Universal Robots PolyScope program: AG_touchoff_demo_tcp.urp

Program AG_touchoff_demo_tcp (installation=AutoGrind directory=/programs/AutoGrind createdIn=5.9.1.1031110 lastSavedIn=5.9.1.1031110 robotSerialNumber=20195501059)
Calibrated DH parameters: a=[0.000146, -0.418764, -0.053981, 0.000058, -0.000023, 0]; d=[0.162545, 37.319448, -206.067439, 168.881546, 0.09955, 0.099464]; alpha=[1.57004, -0.001979, 0.002304, 1.570607, -1.57066, 0]; deltaTheta=[0, -0.174616, -1.258233, 1.432844, -0.000001, 0]
BeforeStart
  start_p := get_actual_tcp_pose()
  MoveJ speed 60 deg/s, acceleration 80 deg/s^2 (useActiveTCP=true) feature=Base
    Waypoint Waypoint (Variable): variable=start_p
  SuppressedNode
    MoveL speed 250 mm/s, acceleration 1200 mm/s^2 (useActiveTCP=true) feature=Base
      Waypoint touch_p: TCP in base x=139.318 y=-525.776 z=17.202 mm, rx=0.0001 ry=0 rz=0.0079 rad; joints [90.599, -70.237, 113.873, -133.625, -89.96, 180.189] deg; TCP offset x=0 y=0 z=175 mm, rx=-3.1416 ry=0 rz=0 rad
Robot Program (runOnlyOnce=true)
  MoveL speed 250 mm/s, acceleration 1200 mm/s^2 (useActiveTCP=true) feature=Base
    MoveDirectionNode (selectedDirection=ZPlus toolParams=0.02, 0.5) feature=Joint_6_name
      Until TOOL_CONTACT_DETECTION (allowActions=false retraction=0.001 decelerationAcceleration=1 decelerationAngularAcceleration=34.906585)
      Until DISTANCE (allowActions=true deceleration=3 distanceNodeType=STOP) Distance=0.025; motionParameters(blendRadius=0)
        Popup Message (haltProgram=false message=No part encountered inputType=Text)
